(* Logix 5000 project; controller WP_Ottawa_Data_Concentrator_1 vendor 1 type 14 code 167 rev 32.14; software revision 32.04; part 3 of 5 *)
(* tags used below, declared in another part *)
   Break_1stStation : BOOL;
   Break_LineWide : BOOL;
   Break_WorkCenter : BOOL;
   Break_Workstation : BOOL;
   LN31_1st_Station_Break_Code : DINT;
   LN31_Assembly_MNT : DINT;
   LN31_Blocked_At_Run_Test_Exit : DINT;
   LN31_Blocked_By_Penske_CAL : DINT;
   LN31_Blocked_By_Repair : DINT;
   LN31_Blocked_By_Wrapper : DINT;
   LN31_BrazingArea_MNT : DINT;
   LN31_Charge_MNT : DINT;
   LN31_CompressorInstall_MNT : DINT;
   LN31_DowntimeCodesMachineA : DINT[120];
   LN31_DowntimeCodesMachineB : DINT[120];
   LN31_DowntimeCodesMachineC : DINT[120];
   LN31_DowntimeCodesMachineD : DINT[120];
   LN31_DowntimeCodesMachineE : DINT[120];
   LN31_DowntimeCodesMachineF : DINT[120];
   LN31_DowntimeCodesMachineG : DINT[120];
   LN31_DowntimeCodesMachineH : DINT[120];
   LN31_DowntimeCodesMachineI : DINT[120];
   LN31_DowntimeCodesMachineOA : DINT[120];
   LN31_DowntimeCodesMachineX : DINT[120];
   LN31_EStop_HMI1 : DINT;
   LN31_EStop_HMI2 : DINT;
   LN31_EStop_Main_Panel : DINT;
   LN31_EStop_Remote_Panel : DINT;
   LN31_EvacLoop_MNT : DINT;
   LN31_FPY : REAL;
   LN31_Ignition_NewSNModel : BOOL[32];
   LN31_Ignition_SNModelMSG : STRING[5];
   LN31_InspectionAndTest_MNT : DINT;
   LN31_Kit_Zone_1_Exit_Fault : DINT;
   LN31_Kitting_MNT : DINT;
   LN31_Label_Machines_Faulted : DINT;
   LN31_Label_Missing : DINT;
   LN31_MachineOverAll_MNT : DINT;
   LN31_Messages_Barcode_SNModel : Barcode_SNModel;
   LN31_Miscellaneous_MNT : DINT;
   LN31_MLC_Downtime : BOOL;
   LN31_Packout_MNT : DINT;
   LN31_PrefoamGlueAndFoam_MNT : DINT;
   LN31_Schedule : UDT_Current_Status;
   LN31_Starved_By_Surge : DINT;
   LN31_Surge_Gate_Open : DINT;
   LN31_WorkstationsA : DINT[120];
   LN31_WorkstationsB : DINT[120];
   LN31_WorkstationsC : DINT[120];
   LN31_WorkstationsD : DINT[120];
   LN31_WorkstationsE : DINT[120];
   LN31_WorkstationsF : DINT[120];
   LN31_WorkstationsG : DINT[120];
   LN31_WorkstationsH : DINT[120];
   LN31_WorkstationsI : DINT[120];
   LN31_WorkstationsOA : DINT[120];
   LN31_WorkstationsX : DINT[120];
   LN31_Wrong_Compressor : DINT;
   LN31_Z22F_Over_Cycle_Time : DINT;
   LN31EAM02 : DINT;
   LN31EAM03 : DINT;
   LN31EFM01 : DINT;
   LN31EFM02 : DINT;
   LN31EFM03 : DINT;
   LN31EGM01 : DINT;
   LN31EGM02 : DINT;
   LN31EGM03 : DINT;
   LN31EGM04 : DINT;
   LN31EHS01 : DINT;
   LN31EHS02 : DINT;
   LN31EHS03 : DINT;
   LN31EHS04 : DINT;
   LN31EHS05 : DINT;
   LN31EHS06 : DINT;
   LN31EHS07 : DINT;
   LN31EHS08 : DINT;
   LN31EIS05 : DINT;
   LN31NCM02 : DINT;
   LN31NDM01 : DINT;
   LN31NDM02 : DINT;
   LN31NDM03 : DINT;
   LN31NIS02 : DINT;
   LN31NIS03 : DINT;
   LN31NIS04 : DINT;
   LN31NIS06 : DINT;
   LN31NIS07 : DINT;
   LN31NIS08 : DINT;
   LN31NIS09 : DINT;
   LN31NIS10 : DINT;
   LN31NIS11 : DINT;
   LN31NIS12 : DINT;
   LN31NIS13 : DINT;
   LN31NIS14 : DINT;
   LN31NIS15 : DINT;
   LN31NIS16 : DINT;
   LN31NIS17 : DINT;
   LN31SBM01 : DINT;
   LN31SBM02 : DINT;
   LN31SBM03 : DINT;
   LN31SBM04 : DINT;
   LN31SBM05 : DINT;
   LN31SCM01 : DINT;
   LN31SDM03 : DINT;
   LN31SIS02 : DINT;
   LN31SIS06 : DINT;
   LN31WAM01 : DINT;
   LN31WAM02 : DINT;
   LN31WEM01 : DINT;
   LN31WEM02 : DINT;
   LN31WEM03 : DINT;
   LN31WEM04 : DINT;
   LN31WEM05 : DINT;
   LN31WEM06 : DINT;
   LN31WEM07 : DINT;
   LN31WEM08 : DINT;
   LN31WEM09 : DINT;
   LN31WFM01 : DINT;
   LN31WFM02 : DINT;
   LN31WFM03 : DINT;
   LN31WGM02 : DINT;
   LN31WGM04 : DINT;
   LN31WIS01 : DINT;
   LN31XAM01 : DINT;
   LN31XAM02 : DINT;
   LN31XAS01 : DINT;
   LN31XAS02 : DINT;
   LN31XBM01 : DINT;
   LN31XBM02 : DINT;
(* LN31, continued *)

ROUTINE R03_DataFromLines   (* ladder *)
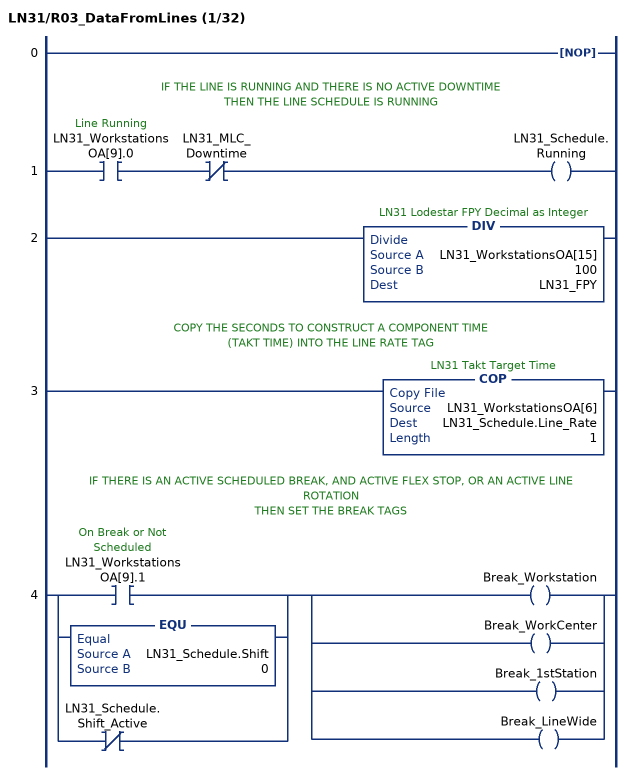
   0: NOP();
   // IF THE LINE IS RUNNING AND THERE IS NO ACTIVE DOWNTIME
   // THEN THE LINE SCHEDULE IS RUNNING
   1: XIC(LN31_WorkstationsOA[9].0)XIO(LN31_MLC_Downtime)OTE(LN31_Schedule.Running);
   2: DIV(LN31_WorkstationsOA[15],100,LN31_FPY);
   // COPY THE SECONDS TO CONSTRUCT A COMPONENT TIME
   // (TAKT TIME) INTO THE LINE RATE TAG
   3: COP(LN31_WorkstationsOA[6],LN31_Schedule.Line_Rate,1);
   // IF THERE IS AN ACTIVE SCHEDULED BREAK, AND ACTIVE FLEX STOP, OR AN ACTIVE LINE ROTATION
   // THEN SET THE BREAK TAGS
   4: [XIC(LN31_WorkstationsOA[9].1) ,EQU(LN31_Schedule.Shift,0) ,XIO(LN31_Schedule.Shift_Active) ][OTE(Break_Workstation) ,OTE(Break_WorkCenter) ,OTE(Break_1stStation) ,OTE(Break_LineWide) ];
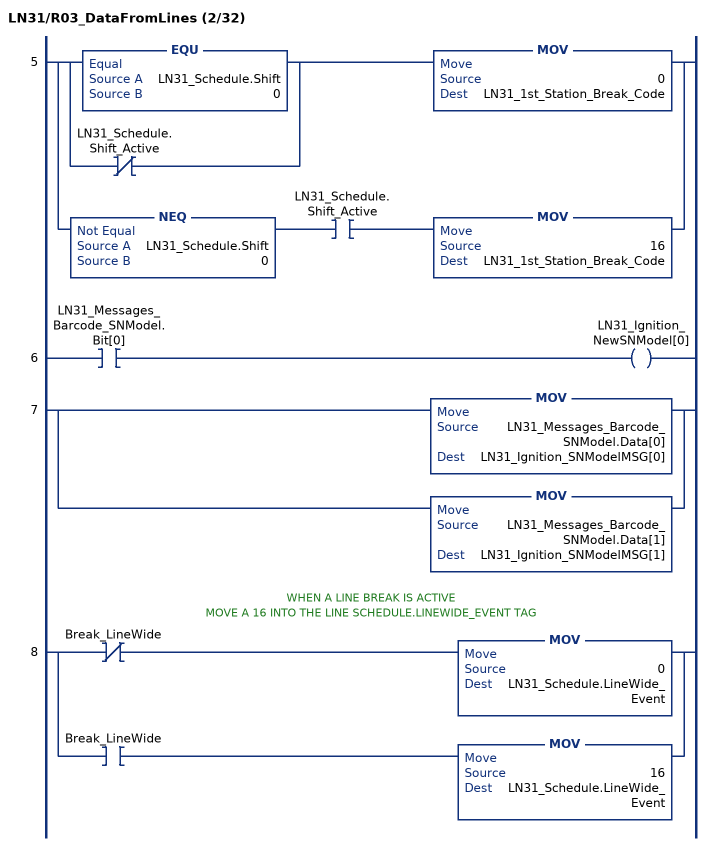
   5: [[EQU(LN31_Schedule.Shift,0) ,XIO(LN31_Schedule.Shift_Active) ] MOV(0,LN31_1st_Station_Break_Code) ,NEQ(LN31_Schedule.Shift,0) XIC(LN31_Schedule.Shift_Active) MOV(16,LN31_1st_Station_Break_Code) ];
   6: XIC(LN31_Messages_Barcode_SNModel.Bit[0])OTE(LN31_Ignition_NewSNModel[0]);
   7: [MOV(LN31_Messages_Barcode_SNModel.Data[0],LN31_Ignition_SNModelMSG[0]) ,MOV(LN31_Messages_Barcode_SNModel.Data[1],LN31_Ignition_SNModelMSG[1]) ];
   // WHEN A LINE BREAK IS ACTIVE
   // MOVE A 16 INTO THE LINE SCHEDULE.LINEWIDE_EVENT TAG
   8: [XIO(Break_LineWide) MOV(0,LN31_Schedule.LineWide_Event) ,XIC(Break_LineWide) MOV(16,LN31_Schedule.LineWide_Event) ];
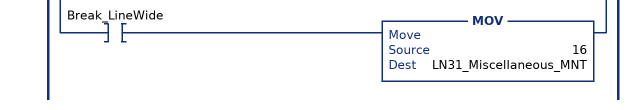
   // MNT Faults
   // If an MNT workcenter is tied to the main line or subline where there is already a workcenter with a workstaiton where "Break_LineWide (when high) MOVEs a 16 in, then that MNT can MOVE a 0 in when "Break_LineWide" goes high
   // If it is an independent MNT (not tied to a workcenter), "Break_LineWide" Tag should MOVE a 16 when "Break_LineWide" goes high
   9: [XIO(Break_LineWide) MOV(LN31_DowntimeCodesMachineA[0],LN31_BrazingArea_MNT) ,XIC(Break_LineWide) MOV(0,LN31_BrazingArea_MNT) ,XIO(Break_LineWide) MOV(LN31_DowntimeCodesMachineB[0],LN31_CompressorInstall_MNT) ,XIC(Break_LineWide) MOV(0,LN31_CompressorInstall_MNT) ,XIO(Break_LineWide) MOV(LN31_DowntimeCodesMachineC[0],LN31_EvacLoop_MNT) ,XIC(Break_LineWide) MOV(0,LN31_EvacLoop_MNT) ,XIO(Break_LineWide) MOV(LN31_DowntimeCodesMachineD[0],LN31_Charge_MNT) ,XIC(Break_LineWide) MOV(0,LN31_Charge_MNT) ,XIO(Break_LineWide) MOV(LN31_DowntimeCodesMachineE[0],LN31_Assembly_MNT) ,XIC(Break_LineWide) MOV(0,LN31_Assembly_MNT) ,XIO(Break_LineWide) MOV(LN31_DowntimeCodesMachineF[0],LN31_InspectionAndTest_MNT) ,XIC(Break_LineWide) MOV(0,LN31_InspectionAndTest_MNT) ,XIO(Break_LineWide) MOV(LN31_DowntimeCodesMachineG[0],LN31_Packout_MNT) ,XIC(Break_LineWide) MOV(0,LN31_Packout_MNT) ,XIO(Break_LineWide) MOV(LN31_DowntimeCodesMachineH[0],LN31_Kitting_MNT) ,XIC(Break_LineWide) MOV(0,LN31_Kitting_MNT) ,XIO(Break_LineWide) MOV(LN31_DowntimeCodesMachineI[0],LN31_PrefoamGlueAndFoam_MNT) ,XIC(Break_LineWide) MOV(16,LN31_PrefoamGlueAndFoam_MNT) ,XIO(Break_LineWide) MOV(LN31_DowntimeCodesMachineOA[0],LN31_MachineOverAll_MNT) ,XIC(Break_LineWide) MOV(0,LN31_MachineOverAll_MNT) ,XIO(Break_LineWide) MOV(LN31_DowntimeCodesMachineX[0],LN31_Miscellaneous_MNT) ,XIC(Break_LineWide) MOV(16,LN31_Miscellaneous_MNT) ];
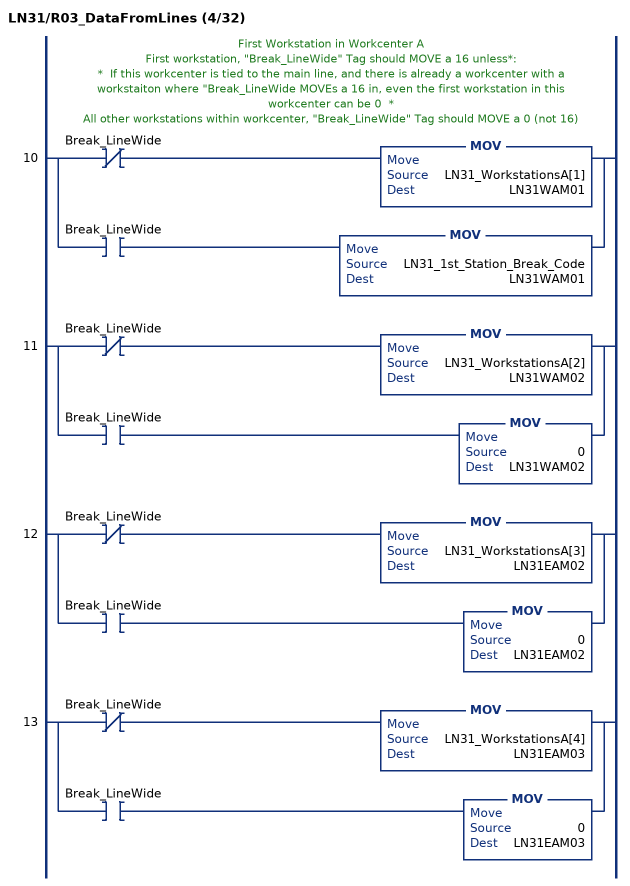
   // First Workstation in Workcenter A
   // First workstation, "Break_LineWide" Tag should MOVE a 16 unless*:
   // *  If this workcenter is tied to the main line, and there is already a workcenter with a workstaiton where "Break_LineWide MOVEs a 16 in, even the first workstation in this workcenter can be 0  *
   // All other workstations within workcenter, "Break_LineWide" Tag should MOVE a 0 (not 16)
   10: [XIO(Break_LineWide) MOV(LN31_WorkstationsA[1],LN31WAM01) ,XIC(Break_LineWide) MOV(LN31_1st_Station_Break_Code,LN31WAM01) ];
   11: [XIO(Break_LineWide) MOV(LN31_WorkstationsA[2],LN31WAM02) ,XIC(Break_LineWide) MOV(0,LN31WAM02) ];
   12: [XIO(Break_LineWide) MOV(LN31_WorkstationsA[3],LN31EAM02) ,XIC(Break_LineWide) MOV(0,LN31EAM02) ];
   13: [XIO(Break_LineWide) MOV(LN31_WorkstationsA[4],LN31EAM03) ,XIC(Break_LineWide) MOV(0,LN31EAM03) ];
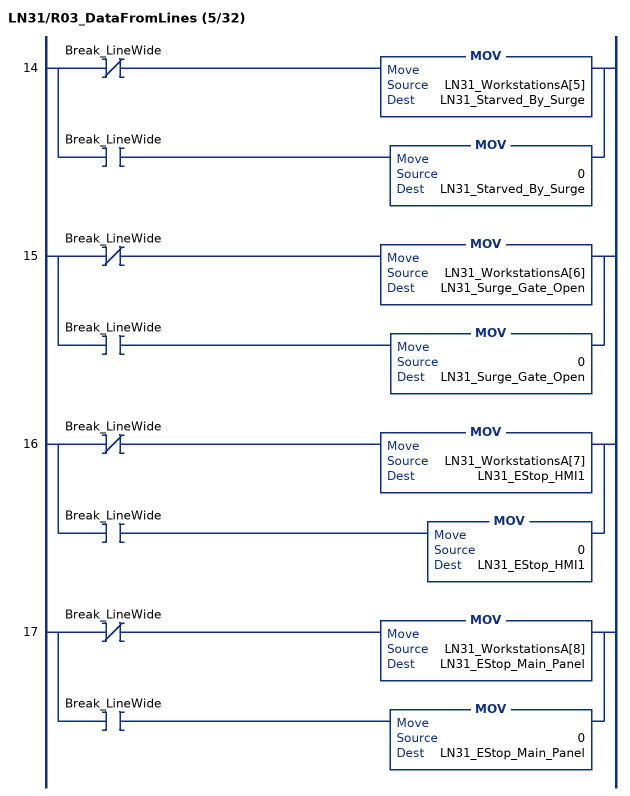
   14: [XIO(Break_LineWide) MOV(LN31_WorkstationsA[5],LN31_Starved_By_Surge) ,XIC(Break_LineWide) MOV(0,LN31_Starved_By_Surge) ];
   15: [XIO(Break_LineWide) MOV(LN31_WorkstationsA[6],LN31_Surge_Gate_Open) ,XIC(Break_LineWide) MOV(0,LN31_Surge_Gate_Open) ];
   16: [XIO(Break_LineWide) MOV(LN31_WorkstationsA[7],LN31_EStop_HMI1) ,XIC(Break_LineWide) MOV(0,LN31_EStop_HMI1) ];
   17: [XIO(Break_LineWide) MOV(LN31_WorkstationsA[8],LN31_EStop_Main_Panel) ,XIC(Break_LineWide) MOV(0,LN31_EStop_Main_Panel) ];
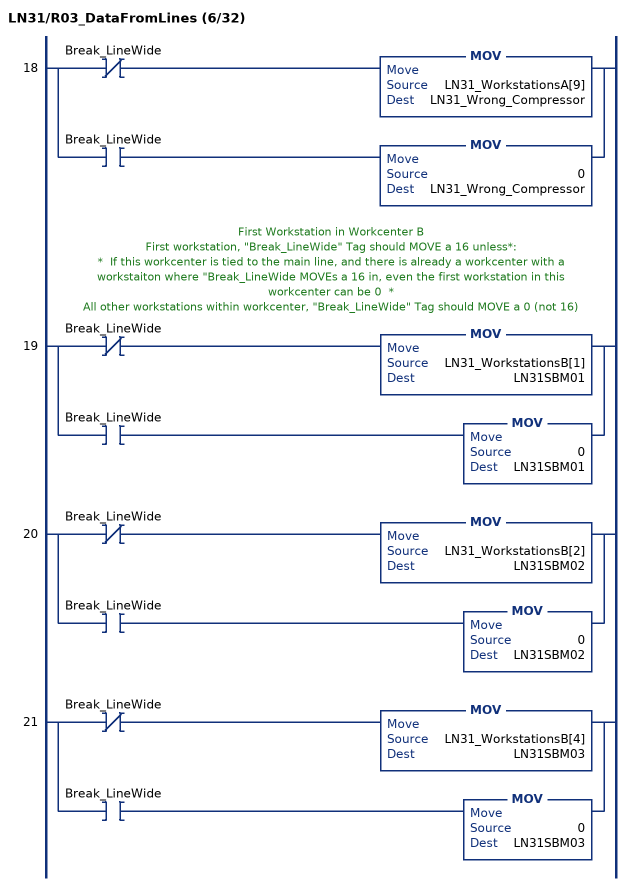
   18: [XIO(Break_LineWide) MOV(LN31_WorkstationsA[9],LN31_Wrong_Compressor) ,XIC(Break_LineWide) MOV(0,LN31_Wrong_Compressor) ];
   // First Workstation in Workcenter B
   // First workstation, "Break_LineWide" Tag should MOVE a 16 unless*:
   // *  If this workcenter is tied to the main line, and there is already a workcenter with a workstaiton where "Break_LineWide MOVEs a 16 in, even the first workstation in this workcenter can be 0  *
   // All other workstations within workcenter, "Break_LineWide" Tag should MOVE a 0 (not 16)
   19: [XIO(Break_LineWide) MOV(LN31_WorkstationsB[1],LN31SBM01) ,XIC(Break_LineWide) MOV(0,LN31SBM01) ];
   20: [XIO(Break_LineWide) MOV(LN31_WorkstationsB[2],LN31SBM02) ,XIC(Break_LineWide) MOV(0,LN31SBM02) ];
   21: [XIO(Break_LineWide) MOV(LN31_WorkstationsB[4],LN31SBM03) ,XIC(Break_LineWide) MOV(0,LN31SBM03) ];
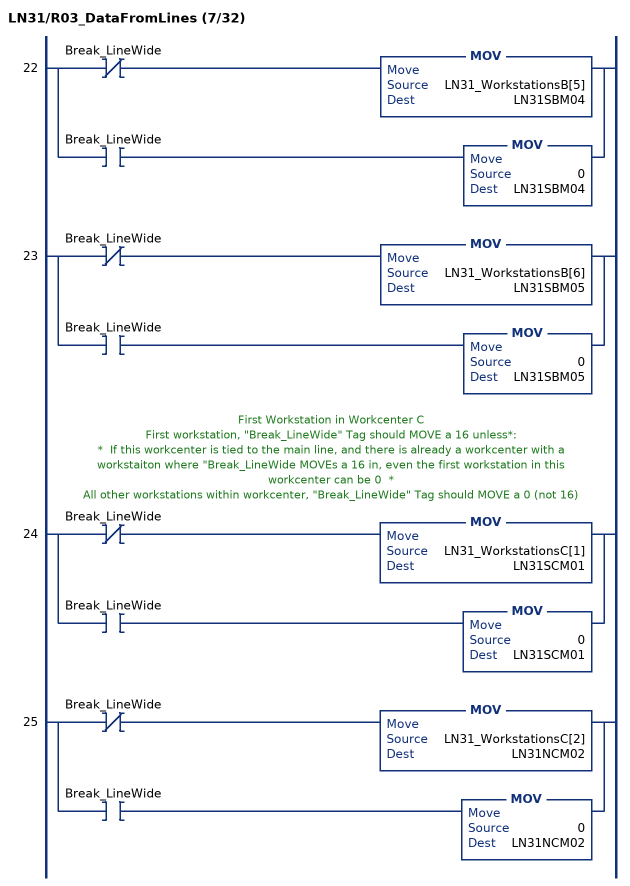
   22: [XIO(Break_LineWide) MOV(LN31_WorkstationsB[5],LN31SBM04) ,XIC(Break_LineWide) MOV(0,LN31SBM04) ];
   23: [XIO(Break_LineWide) MOV(LN31_WorkstationsB[6],LN31SBM05) ,XIC(Break_LineWide) MOV(0,LN31SBM05) ];
   // First Workstation in Workcenter C
   // First workstation, "Break_LineWide" Tag should MOVE a 16 unless*:
   // *  If this workcenter is tied to the main line, and there is already a workcenter with a workstaiton where "Break_LineWide MOVEs a 16 in, even the first workstation in this workcenter can be 0  *
   // All other workstations within workcenter, "Break_LineWide" Tag should MOVE a 0 (not 16)
   24: [XIO(Break_LineWide) MOV(LN31_WorkstationsC[1],LN31SCM01) ,XIC(Break_LineWide) MOV(0,LN31SCM01) ];
   25: [XIO(Break_LineWide) MOV(LN31_WorkstationsC[2],LN31NCM02) ,XIC(Break_LineWide) MOV(0,LN31NCM02) ];
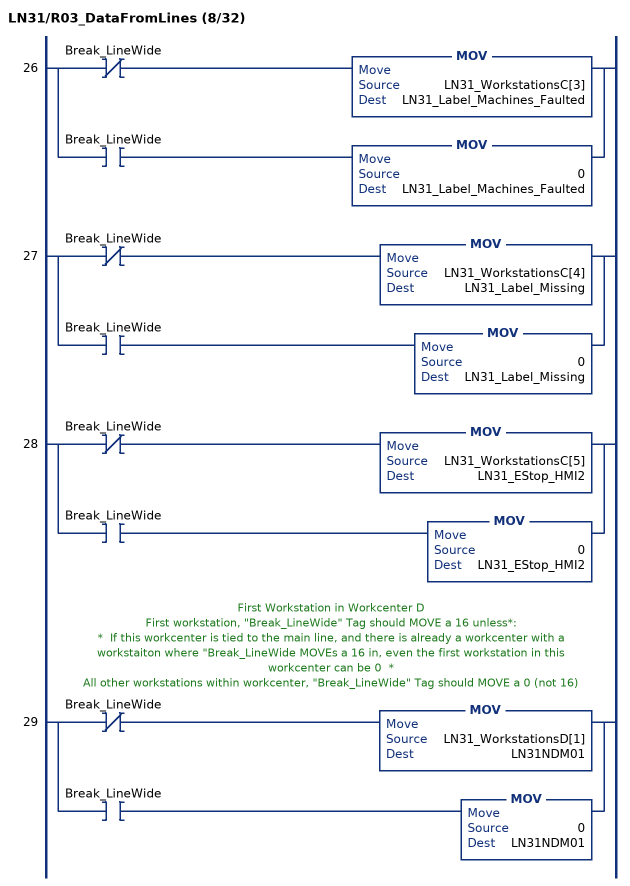
   26: [XIO(Break_LineWide) MOV(LN31_WorkstationsC[3],LN31_Label_Machines_Faulted) ,XIC(Break_LineWide) MOV(0,LN31_Label_Machines_Faulted) ];
   27: [XIO(Break_LineWide) MOV(LN31_WorkstationsC[4],LN31_Label_Missing) ,XIC(Break_LineWide) MOV(0,LN31_Label_Missing) ];
   28: [XIO(Break_LineWide) MOV(LN31_WorkstationsC[5],LN31_EStop_HMI2) ,XIC(Break_LineWide) MOV(0,LN31_EStop_HMI2) ];
   // First Workstation in Workcenter D
   // First workstation, "Break_LineWide" Tag should MOVE a 16 unless*:
   // *  If this workcenter is tied to the main line, and there is already a workcenter with a workstaiton where "Break_LineWide MOVEs a 16 in, even the first workstation in this workcenter can be 0  *
   // All other workstations within workcenter, "Break_LineWide" Tag should MOVE a 0 (not 16)
   29: [XIO(Break_LineWide) MOV(LN31_WorkstationsD[1],LN31NDM01) ,XIC(Break_LineWide) MOV(0,LN31NDM01) ];
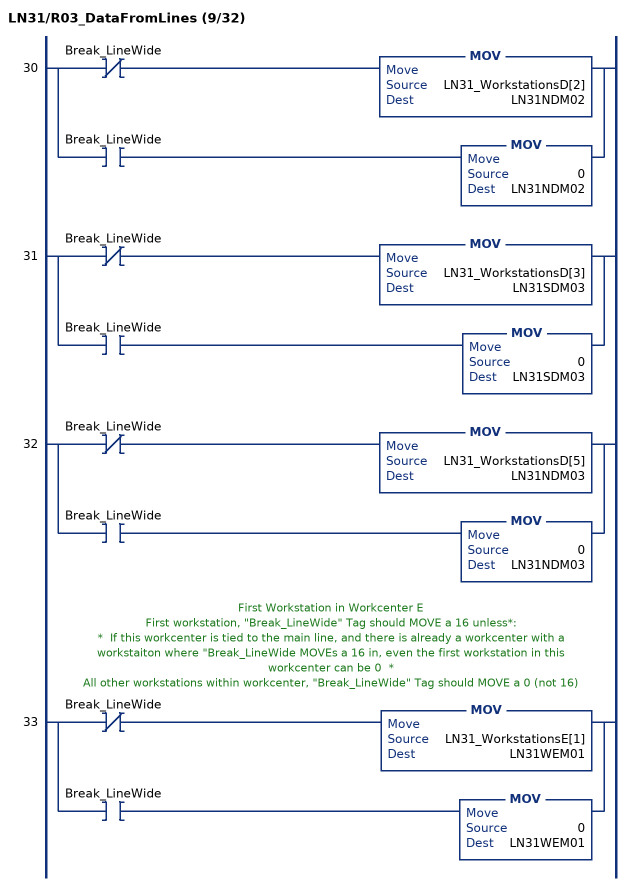
   30: [XIO(Break_LineWide) MOV(LN31_WorkstationsD[2],LN31NDM02) ,XIC(Break_LineWide) MOV(0,LN31NDM02) ];
   31: [XIO(Break_LineWide) MOV(LN31_WorkstationsD[3],LN31SDM03) ,XIC(Break_LineWide) MOV(0,LN31SDM03) ];
   32: [XIO(Break_LineWide) MOV(LN31_WorkstationsD[5],LN31NDM03) ,XIC(Break_LineWide) MOV(0,LN31NDM03) ];
   // First Workstation in Workcenter E
   // First workstation, "Break_LineWide" Tag should MOVE a 16 unless*:
   // *  If this workcenter is tied to the main line, and there is already a workcenter with a workstaiton where "Break_LineWide MOVEs a 16 in, even the first workstation in this workcenter can be 0  *
   // All other workstations within workcenter, "Break_LineWide" Tag should MOVE a 0 (not 16)
   33: [XIO(Break_LineWide) MOV(LN31_WorkstationsE[1],LN31WEM01) ,XIC(Break_LineWide) MOV(0,LN31WEM01) ];
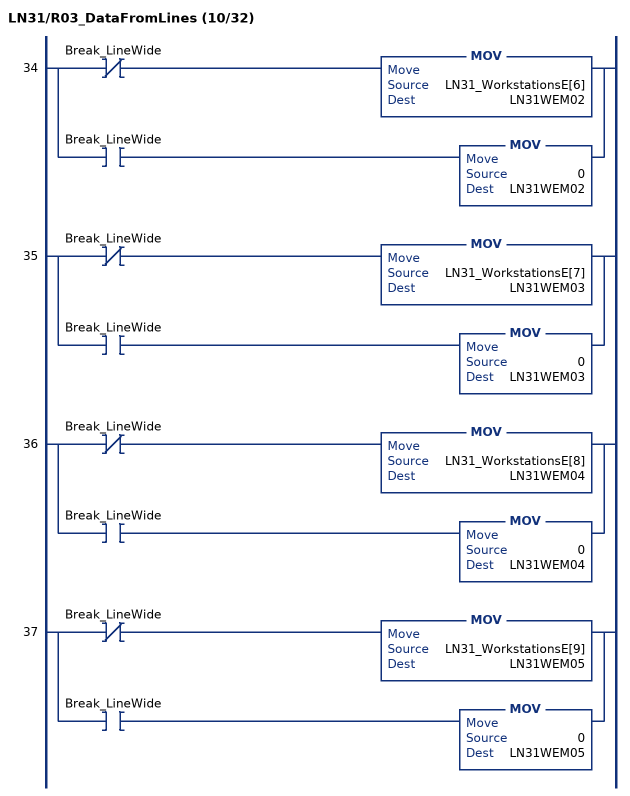
   34: [XIO(Break_LineWide) MOV(LN31_WorkstationsE[6],LN31WEM02) ,XIC(Break_LineWide) MOV(0,LN31WEM02) ];
   35: [XIO(Break_LineWide) MOV(LN31_WorkstationsE[7],LN31WEM03) ,XIC(Break_LineWide) MOV(0,LN31WEM03) ];
   36: [XIO(Break_LineWide) MOV(LN31_WorkstationsE[8],LN31WEM04) ,XIC(Break_LineWide) MOV(0,LN31WEM04) ];
   37: [XIO(Break_LineWide) MOV(LN31_WorkstationsE[9],LN31WEM05) ,XIC(Break_LineWide) MOV(0,LN31WEM05) ];
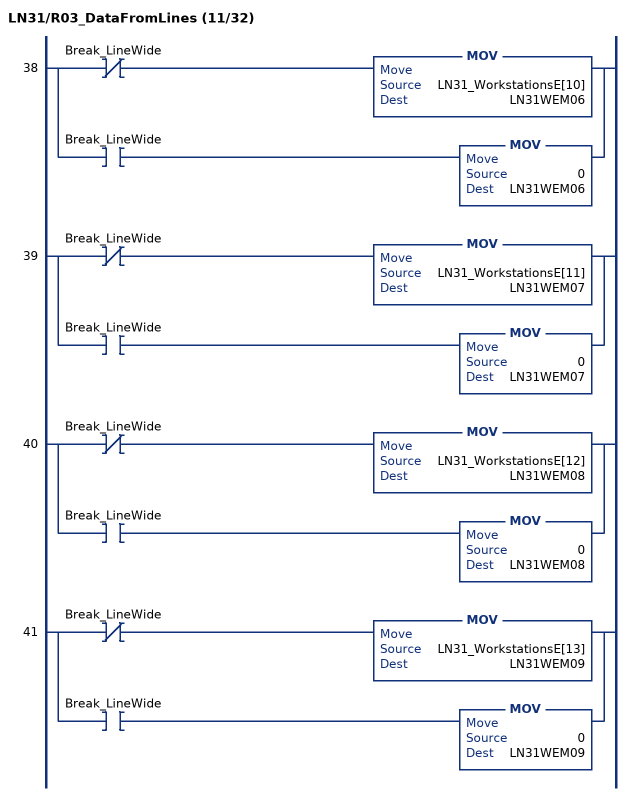
   38: [XIO(Break_LineWide) MOV(LN31_WorkstationsE[10],LN31WEM06) ,XIC(Break_LineWide) MOV(0,LN31WEM06) ];
   39: [XIO(Break_LineWide) MOV(LN31_WorkstationsE[11],LN31WEM07) ,XIC(Break_LineWide) MOV(0,LN31WEM07) ];
   40: [XIO(Break_LineWide) MOV(LN31_WorkstationsE[12],LN31WEM08) ,XIC(Break_LineWide) MOV(0,LN31WEM08) ];
   41: [XIO(Break_LineWide) MOV(LN31_WorkstationsE[13],LN31WEM09) ,XIC(Break_LineWide) MOV(0,LN31WEM09) ];
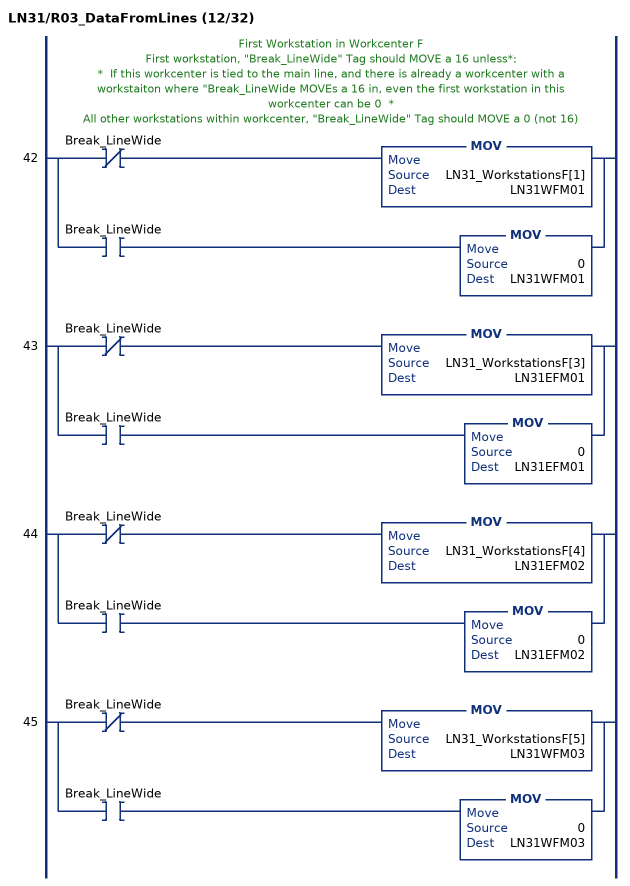
   // First Workstation in Workcenter F
   // First workstation, "Break_LineWide" Tag should MOVE a 16 unless*:
   // *  If this workcenter is tied to the main line, and there is already a workcenter with a workstaiton where "Break_LineWide MOVEs a 16 in, even the first workstation in this workcenter can be 0  *
   // All other workstations within workcenter, "Break_LineWide" Tag should MOVE a 0 (not 16)
   42: [XIO(Break_LineWide) MOV(LN31_WorkstationsF[1],LN31WFM01) ,XIC(Break_LineWide) MOV(0,LN31WFM01) ];
   43: [XIO(Break_LineWide) MOV(LN31_WorkstationsF[3],LN31EFM01) ,XIC(Break_LineWide) MOV(0,LN31EFM01) ];
   44: [XIO(Break_LineWide) MOV(LN31_WorkstationsF[4],LN31EFM02) ,XIC(Break_LineWide) MOV(0,LN31EFM02) ];
   45: [XIO(Break_LineWide) MOV(LN31_WorkstationsF[5],LN31WFM03) ,XIC(Break_LineWide) MOV(0,LN31WFM03) ];
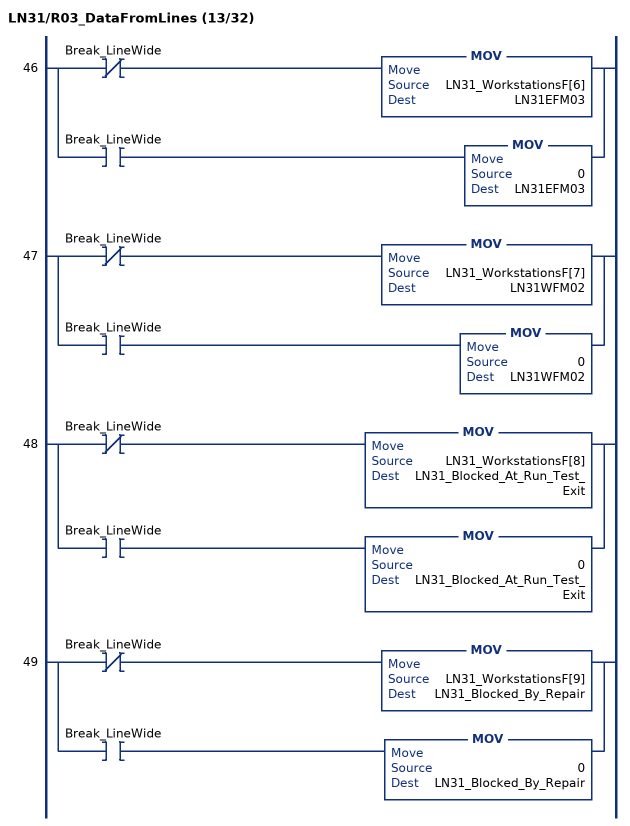
   46: [XIO(Break_LineWide) MOV(LN31_WorkstationsF[6],LN31EFM03) ,XIC(Break_LineWide) MOV(0,LN31EFM03) ];
   47: [XIO(Break_LineWide) MOV(LN31_WorkstationsF[7],LN31WFM02) ,XIC(Break_LineWide) MOV(0,LN31WFM02) ];
   48: [XIO(Break_LineWide) MOV(LN31_WorkstationsF[8],LN31_Blocked_At_Run_Test_Exit) ,XIC(Break_LineWide) MOV(0,LN31_Blocked_At_Run_Test_Exit) ];
   49: [XIO(Break_LineWide) MOV(LN31_WorkstationsF[9],LN31_Blocked_By_Repair) ,XIC(Break_LineWide) MOV(0,LN31_Blocked_By_Repair) ];
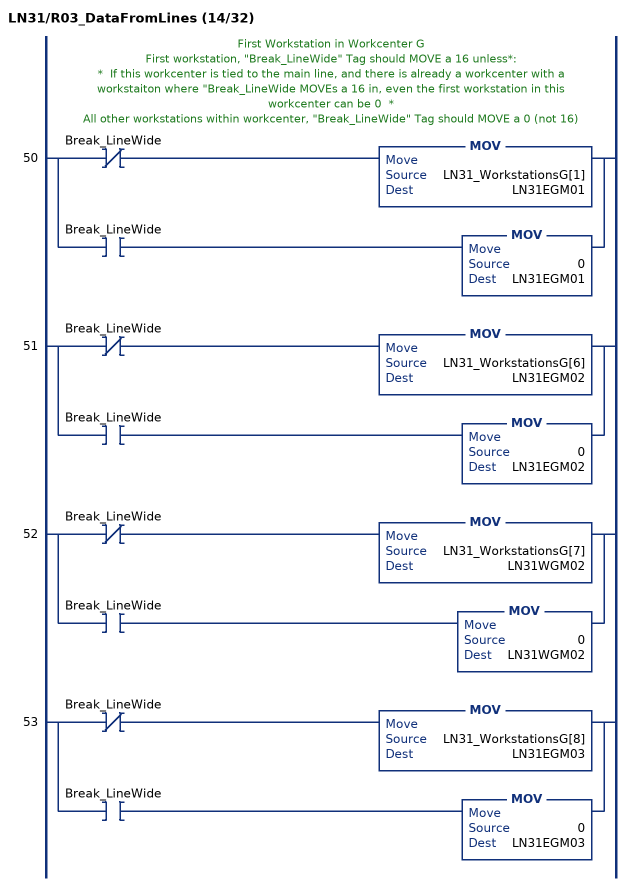
   // First Workstation in Workcenter G
   // First workstation, "Break_LineWide" Tag should MOVE a 16 unless*:
   // *  If this workcenter is tied to the main line, and there is already a workcenter with a workstaiton where "Break_LineWide MOVEs a 16 in, even the first workstation in this workcenter can be 0  *
   // All other workstations within workcenter, "Break_LineWide" Tag should MOVE a 0 (not 16)
   50: [XIO(Break_LineWide) MOV(LN31_WorkstationsG[1],LN31EGM01) ,XIC(Break_LineWide) MOV(0,LN31EGM01) ];
   51: [XIO(Break_LineWide) MOV(LN31_WorkstationsG[6],LN31EGM02) ,XIC(Break_LineWide) MOV(0,LN31EGM02) ];
   52: [XIO(Break_LineWide) MOV(LN31_WorkstationsG[7],LN31WGM02) ,XIC(Break_LineWide) MOV(0,LN31WGM02) ];
   53: [XIO(Break_LineWide) MOV(LN31_WorkstationsG[8],LN31EGM03) ,XIC(Break_LineWide) MOV(0,LN31EGM03) ];
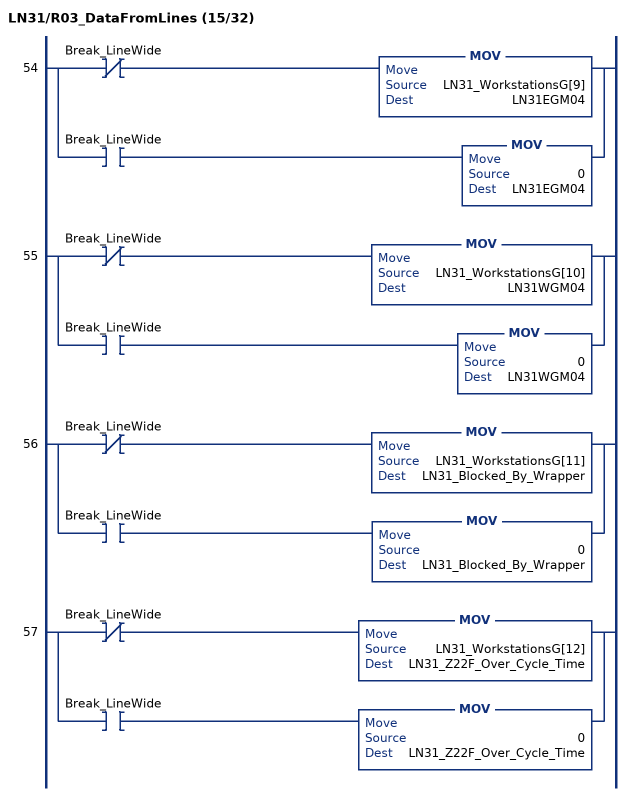
   54: [XIO(Break_LineWide) MOV(LN31_WorkstationsG[9],LN31EGM04) ,XIC(Break_LineWide) MOV(0,LN31EGM04) ];
   55: [XIO(Break_LineWide) MOV(LN31_WorkstationsG[10],LN31WGM04) ,XIC(Break_LineWide) MOV(0,LN31WGM04) ];
   56: [XIO(Break_LineWide) MOV(LN31_WorkstationsG[11],LN31_Blocked_By_Wrapper) ,XIC(Break_LineWide) MOV(0,LN31_Blocked_By_Wrapper) ];
   57: [XIO(Break_LineWide) MOV(LN31_WorkstationsG[12],LN31_Z22F_Over_Cycle_Time) ,XIC(Break_LineWide) MOV(0,LN31_Z22F_Over_Cycle_Time) ];
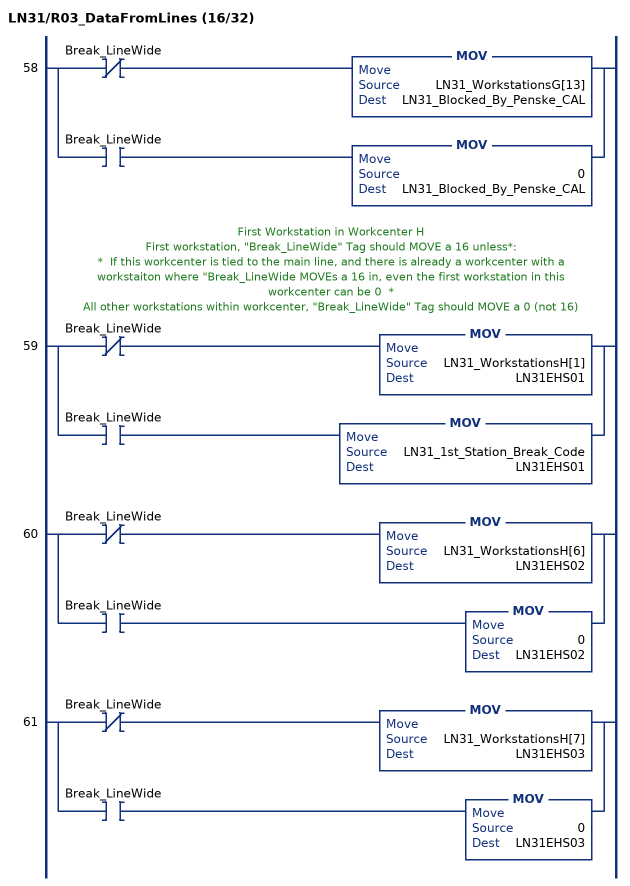
   58: [XIO(Break_LineWide) MOV(LN31_WorkstationsG[13],LN31_Blocked_By_Penske_CAL) ,XIC(Break_LineWide) MOV(0,LN31_Blocked_By_Penske_CAL) ];
   // First Workstation in Workcenter H
   // First workstation, "Break_LineWide" Tag should MOVE a 16 unless*:
   // *  If this workcenter is tied to the main line, and there is already a workcenter with a workstaiton where "Break_LineWide MOVEs a 16 in, even the first workstation in this workcenter can be 0  *
   // All other workstations within workcenter, "Break_LineWide" Tag should MOVE a 0 (not 16)
   59: [XIO(Break_LineWide) MOV(LN31_WorkstationsH[1],LN31EHS01) ,XIC(Break_LineWide) MOV(LN31_1st_Station_Break_Code,LN31EHS01) ];
   60: [XIO(Break_LineWide) MOV(LN31_WorkstationsH[6],LN31EHS02) ,XIC(Break_LineWide) MOV(0,LN31EHS02) ];
   61: [XIO(Break_LineWide) MOV(LN31_WorkstationsH[7],LN31EHS03) ,XIC(Break_LineWide) MOV(0,LN31EHS03) ];
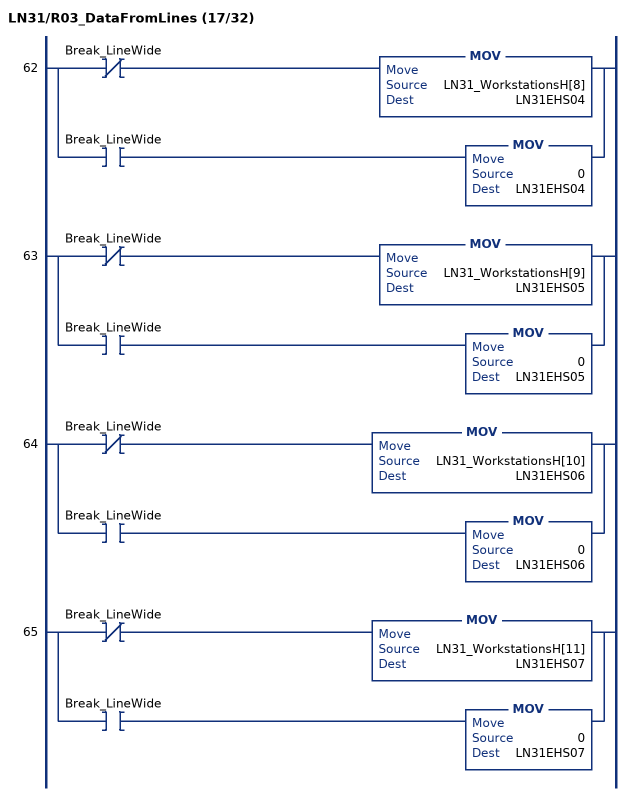
   62: [XIO(Break_LineWide) MOV(LN31_WorkstationsH[8],LN31EHS04) ,XIC(Break_LineWide) MOV(0,LN31EHS04) ];
   63: [XIO(Break_LineWide) MOV(LN31_WorkstationsH[9],LN31EHS05) ,XIC(Break_LineWide) MOV(0,LN31EHS05) ];
   64: [XIO(Break_LineWide) MOV(LN31_WorkstationsH[10],LN31EHS06) ,XIC(Break_LineWide) MOV(0,LN31EHS06) ];
   65: [XIO(Break_LineWide) MOV(LN31_WorkstationsH[11],LN31EHS07) ,XIC(Break_LineWide) MOV(0,LN31EHS07) ];
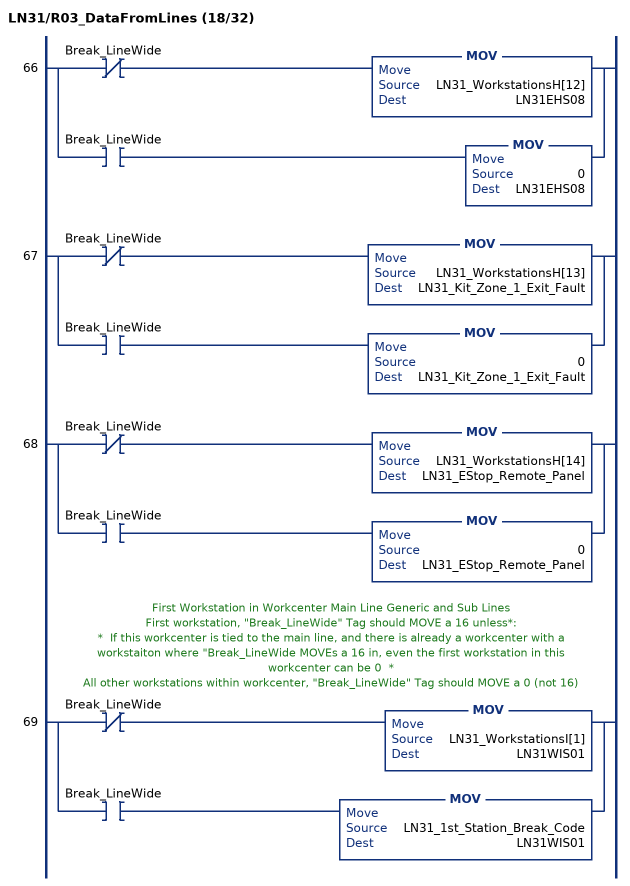
   66: [XIO(Break_LineWide) MOV(LN31_WorkstationsH[12],LN31EHS08) ,XIC(Break_LineWide) MOV(0,LN31EHS08) ];
   67: [XIO(Break_LineWide) MOV(LN31_WorkstationsH[13],LN31_Kit_Zone_1_Exit_Fault) ,XIC(Break_LineWide) MOV(0,LN31_Kit_Zone_1_Exit_Fault) ];
   68: [XIO(Break_LineWide) MOV(LN31_WorkstationsH[14],LN31_EStop_Remote_Panel) ,XIC(Break_LineWide) MOV(0,LN31_EStop_Remote_Panel) ];
   // First Workstation in Workcenter Main Line Generic and Sub Lines
   // First workstation, "Break_LineWide" Tag should MOVE a 16 unless*:
   // *  If this workcenter is tied to the main line, and there is already a workcenter with a workstaiton where "Break_LineWide MOVEs a 16 in, even the first workstation in this workcenter can be 0  *
   // All other workstations within workcenter, "Break_LineWide" Tag should MOVE a 0 (not 16)
   69: [XIO(Break_LineWide) MOV(LN31_WorkstationsI[1],LN31WIS01) ,XIC(Break_LineWide) MOV(LN31_1st_Station_Break_Code,LN31WIS01) ];
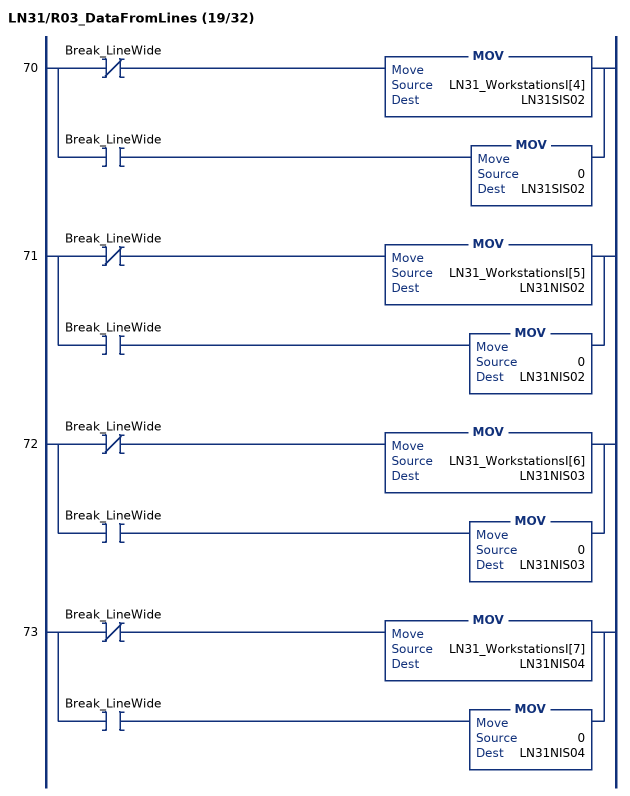
   70: [XIO(Break_LineWide) MOV(LN31_WorkstationsI[4],LN31SIS02) ,XIC(Break_LineWide) MOV(0,LN31SIS02) ];
   71: [XIO(Break_LineWide) MOV(LN31_WorkstationsI[5],LN31NIS02) ,XIC(Break_LineWide) MOV(0,LN31NIS02) ];
   72: [XIO(Break_LineWide) MOV(LN31_WorkstationsI[6],LN31NIS03) ,XIC(Break_LineWide) MOV(0,LN31NIS03) ];
   73: [XIO(Break_LineWide) MOV(LN31_WorkstationsI[7],LN31NIS04) ,XIC(Break_LineWide) MOV(0,LN31NIS04) ];
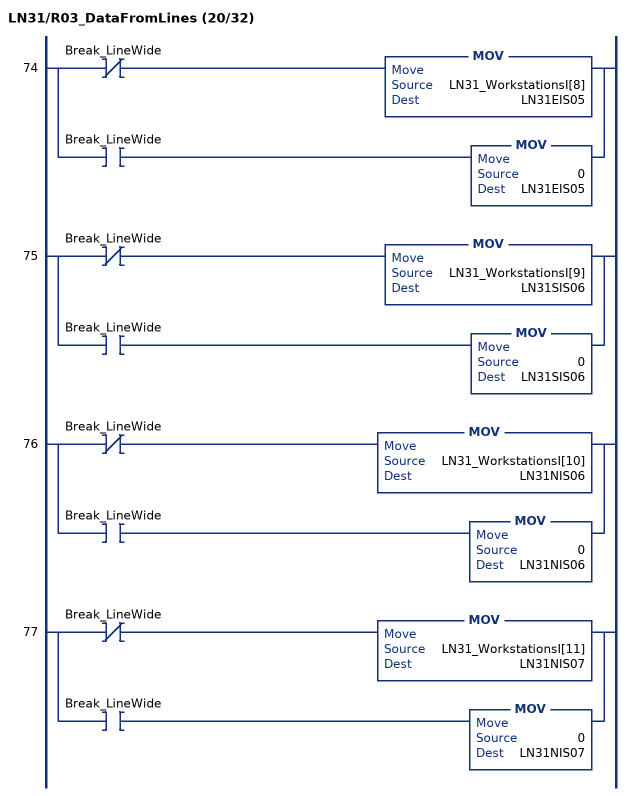
   74: [XIO(Break_LineWide) MOV(LN31_WorkstationsI[8],LN31EIS05) ,XIC(Break_LineWide) MOV(0,LN31EIS05) ];
   75: [XIO(Break_LineWide) MOV(LN31_WorkstationsI[9],LN31SIS06) ,XIC(Break_LineWide) MOV(0,LN31SIS06) ];
   76: [XIO(Break_LineWide) MOV(LN31_WorkstationsI[10],LN31NIS06) ,XIC(Break_LineWide) MOV(0,LN31NIS06) ];
   77: [XIO(Break_LineWide) MOV(LN31_WorkstationsI[11],LN31NIS07) ,XIC(Break_LineWide) MOV(0,LN31NIS07) ];
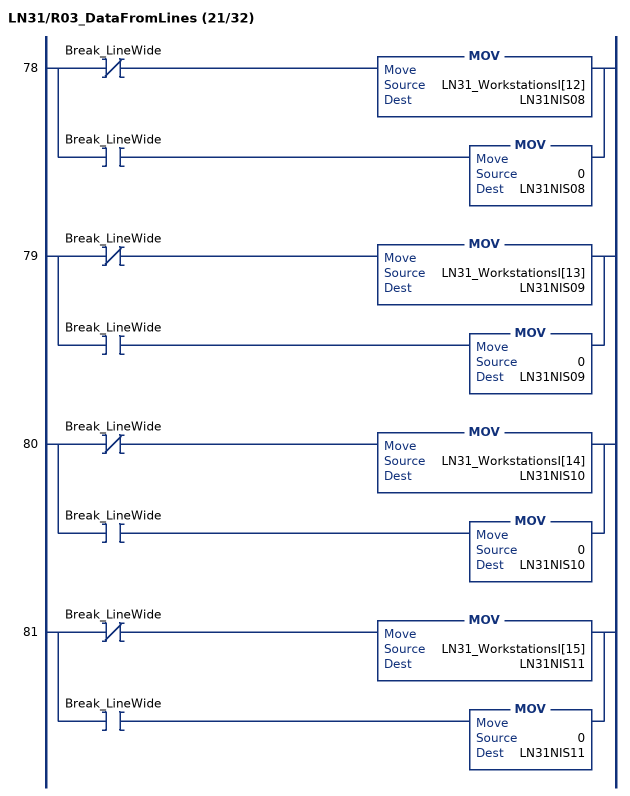
   78: [XIO(Break_LineWide) MOV(LN31_WorkstationsI[12],LN31NIS08) ,XIC(Break_LineWide) MOV(0,LN31NIS08) ];
   79: [XIO(Break_LineWide) MOV(LN31_WorkstationsI[13],LN31NIS09) ,XIC(Break_LineWide) MOV(0,LN31NIS09) ];
   80: [XIO(Break_LineWide) MOV(LN31_WorkstationsI[14],LN31NIS10) ,XIC(Break_LineWide) MOV(0,LN31NIS10) ];
   81: [XIO(Break_LineWide) MOV(LN31_WorkstationsI[15],LN31NIS11) ,XIC(Break_LineWide) MOV(0,LN31NIS11) ];
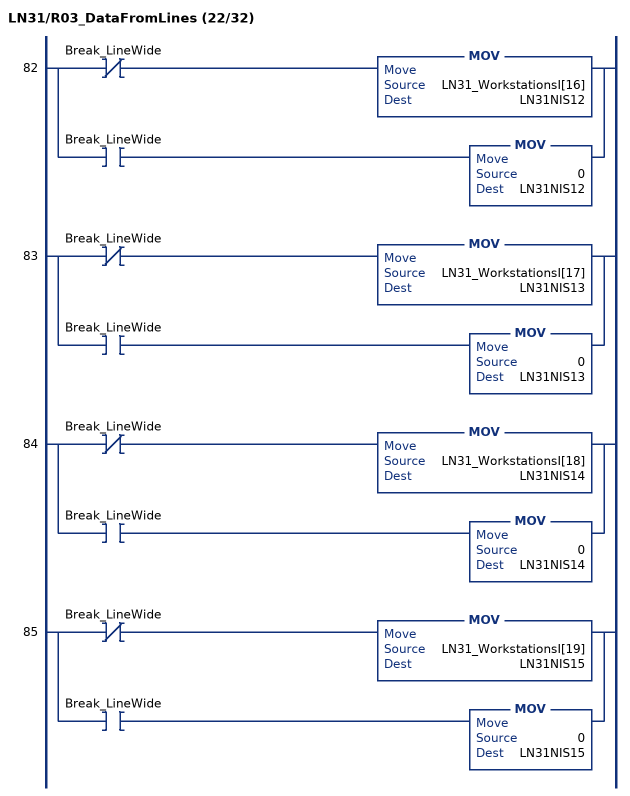
   82: [XIO(Break_LineWide) MOV(LN31_WorkstationsI[16],LN31NIS12) ,XIC(Break_LineWide) MOV(0,LN31NIS12) ];
   83: [XIO(Break_LineWide) MOV(LN31_WorkstationsI[17],LN31NIS13) ,XIC(Break_LineWide) MOV(0,LN31NIS13) ];
   84: [XIO(Break_LineWide) MOV(LN31_WorkstationsI[18],LN31NIS14) ,XIC(Break_LineWide) MOV(0,LN31NIS14) ];
   85: [XIO(Break_LineWide) MOV(LN31_WorkstationsI[19],LN31NIS15) ,XIC(Break_LineWide) MOV(0,LN31NIS15) ];
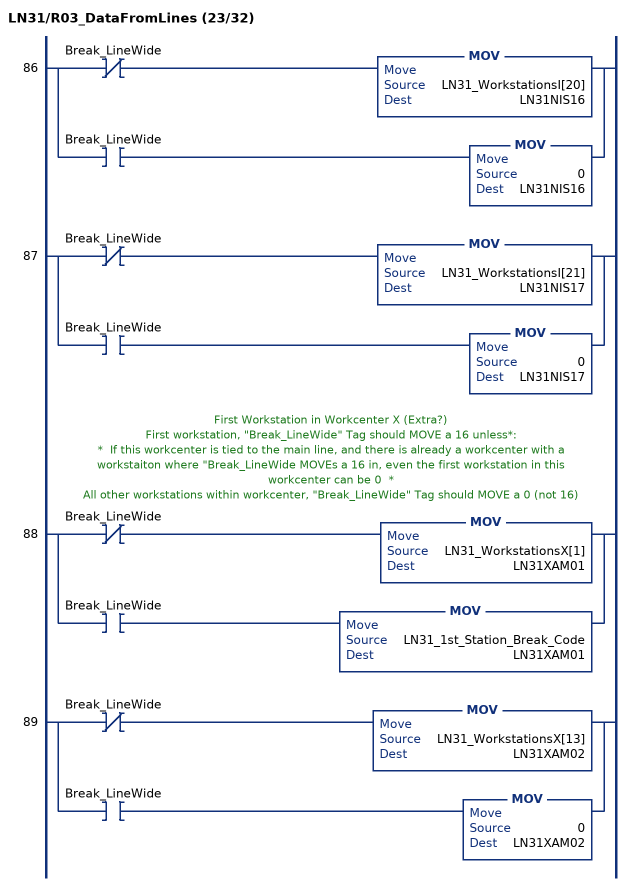
   86: [XIO(Break_LineWide) MOV(LN31_WorkstationsI[20],LN31NIS16) ,XIC(Break_LineWide) MOV(0,LN31NIS16) ];
   87: [XIO(Break_LineWide) MOV(LN31_WorkstationsI[21],LN31NIS17) ,XIC(Break_LineWide) MOV(0,LN31NIS17) ];
   // First Workstation in Workcenter X (Extra?)
   // First workstation, "Break_LineWide" Tag should MOVE a 16 unless*:
   // *  If this workcenter is tied to the main line, and there is already a workcenter with a workstaiton where "Break_LineWide MOVEs a 16 in, even the first workstation in this workcenter can be 0  *
   // All other workstations within workcenter, "Break_LineWide" Tag should MOVE a 0 (not 16)
   88: [XIO(Break_LineWide) MOV(LN31_WorkstationsX[1],LN31XAM01) ,XIC(Break_LineWide) MOV(LN31_1st_Station_Break_Code,LN31XAM01) ];
   89: [XIO(Break_LineWide) MOV(LN31_WorkstationsX[13],LN31XAM02) ,XIC(Break_LineWide) MOV(0,LN31XAM02) ];
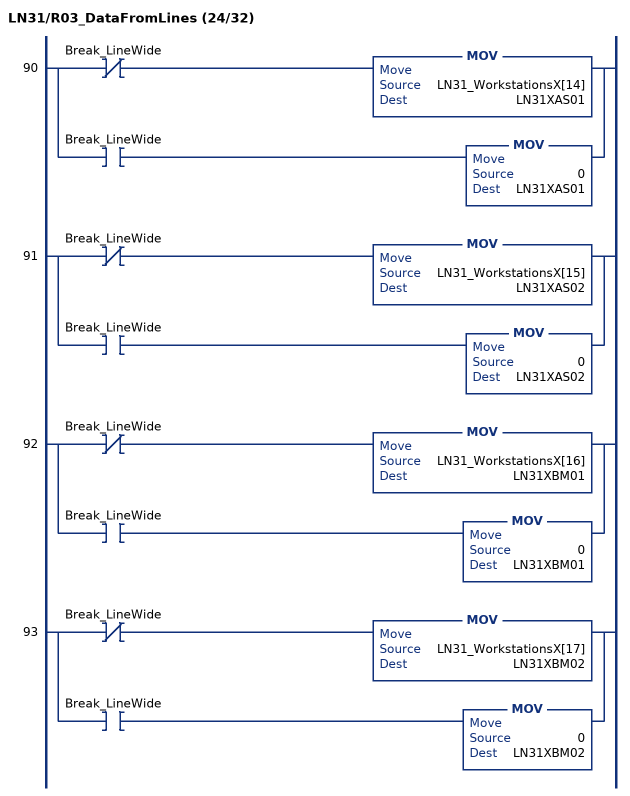
   90: [XIO(Break_LineWide) MOV(LN31_WorkstationsX[14],LN31XAS01) ,XIC(Break_LineWide) MOV(0,LN31XAS01) ];
   91: [XIO(Break_LineWide) MOV(LN31_WorkstationsX[15],LN31XAS02) ,XIC(Break_LineWide) MOV(0,LN31XAS02) ];
   92: [XIO(Break_LineWide) MOV(LN31_WorkstationsX[16],LN31XBM01) ,XIC(Break_LineWide) MOV(0,LN31XBM01) ];
   93: [XIO(Break_LineWide) MOV(LN31_WorkstationsX[17],LN31XBM02) ,XIC(Break_LineWide) MOV(0,LN31XBM02) ];
